Staubli VAL3: computeSequenceDelay.pgx

program computeSequenceDelay(num nLastSequenceSent, num nLastSequenceReceived, num& x_nSequenceDelay)
begin
    x_nSequenceDelay = nLastSequenceSent - nLastSequenceReceived
    // If negative, it means we wrapped around or that there is an error
    if (x_nSequenceDelay < -60000 and x_nSequenceDelay < 0)
      // Wrap around (uint16_t)
      x_nSequenceDelay = x_nSequenceDelay + 65536
    endIf
end
